Fanuc KAREL source: KX00033.KL

PROGRAM KX00033
%NOLOCKGROUP
%UNINITVARS
VAR
  I: INTEGER
  J: INTEGER
  B: BOOLEAN
  F: FILE
  S: STRING[80]
  P: XYZWPR
BEGIN
  I = 1
END KX00033
